Yaskawa INFORM job: FMTV_HOOD_FASH.JBI

/JOB
//NAME FMTV_HOOD_FASH
//POS
///NPOS 40,0,0,0,0,0
///TOOL 0
///POSTYPE PULSE
///PULSE
C00000=-63952,-155163,126853,-105316,-81596,-126671
C00001=-64461,-165808,55284,-105319,-116136,-134897
C00002=-65360,-175099,-71284,-105325,-123848,-149443
C00003=16523,-162142,-76585,-105325,-105920,-149443
C00004=136824,-41147,-71653,-105908,-92109,-42430
C00005=136265,2790,-33985,-105635,-93453,-40514
C00006=131512,-1858,-30509,-105042,-95515,-43185
C00007=137993,-15449,-40810,-106144,-90722,-43513
C00008=137236,-27294,-42795,-96614,-65040,-40742
C00009=140665,-37218,-47628,-99236,-35066,-29992
C00010=140875,-41659,-45027,-77194,-30549,-37243
C00011=146366,-51964,-56030,-75285,-24000,-39354
C00012=156119,-65002,-57409,-21147,-27778,-71904
C00013=185515,-90979,-56740,15089,-40881,-92836
C00014=189457,-94504,-56572,18214,-43459,-94468
C00015=185283,-96154,-47186,13023,-48087,-91295
C00016=200345,-105201,-46417,22564,-56140,-91888
C00017=216925,-109654,-49443,33869,-61566,-97373
C00018=254335,-111877,-36308,-709,-80515,-94448
C00019=248884,-122551,-45515,-3659,-81498,-92809
C00020=231141,-122690,-119580,-13159,-82300,-87441
C00021=-123049,-84648,-100330,119939,-63154,47192
C00022=-145736,-60124,-89141,132014,-54215,37600
C00023=-142792,-13464,-52848,133356,-59585,35650
C00024=-142664,-20455,-52488,131545,-57125,37514
C00025=-150130,-32967,-58116,133370,-50891,37010
C00026=-145449,-39905,-51845,93454,-46937,51672
C00027=-145191,-39750,-50505,88326,-47662,51868
C00028=-144160,-44267,-45166,62771,-52773,58710
C00029=-148791,-53730,-48823,49689,-54914,64885
C00030=-150743,-57181,-50382,48425,-54527,66002
C00031=-175825,-83730,-45254,23478,-63050,83138
C00032=-177177,-85796,-44891,22474,-63852,83945
C00033=-172411,-84272,-42490,25021,-65496,77234
C00034=-167210,-84468,-34339,27016,-70739,76523
C00035=-180047,-97470,-37743,19473,-72177,81934
C00036=-191369,-102527,-40604,12946,-71396,85928
C00037=-242211,-114344,-41149,18289,-76989,98255
C00038=-243523,-126027,-51318,17488,-77632,98803
C00039=-252640,-156391,-84960,58658,-32345,33822
//INST
///DATE 2023/09/19 14:49
///ATTR SC,RW
///GROUP1 RB1
NOP
MOVJ C00000 VJ=65.00  //HOME
MOVJ C00001 VJ=65.00
MOVJ C00002 VJ=65.00  //ROTATE
MOVJ C00003 VJ=65.00
MOVJ C00004 VJ=65.00
MOVL C00005 V=150.0  //OVER
MOVL C00006 V=100.0  //UP TO
MOVL C00007 V=25.0  //INTO
MOVL C00008 V=25.0
MOVL C00009 V=25.0
MOVL C00010 V=25.0
MOVL C00011 V=25.0
MOVL C00012 V=25.0
MOVL C00013 V=25.0
MOVL C00014 V=25.0
MOVL C00015 V=25.0
MOVL C00016 V=25.0
MOVL C00017 V=25.0
MOVL C00018 V=25.0  //END
MOVL C00019 V=45.0  //OUT
MOVJ C00020 VJ=65.00
MOVJ C00021 VJ=65.00
MOVL C00022 V=65.0
MOVL C00023 V=65.0
MOVL C00024 V=65.0  //INLINE
MOVL C00025 V=25.0
MOVL C00026 V=25.0  //CORNER
MOVL C00027 V=10.0
MOVL C00028 V=25.0
MOVL C00029 V=25.0
MOVL C00030 V=25.0
MOVL C00031 V=25.0
MOVL C00032 V=25.0
MOVL C00033 V=25.0
MOVL C00034 V=25.0
MOVL C00035 V=25.0
MOVL C00036 V=25.0
MOVL C00037 V=25.0  //END
MOVJ C00038 VJ=65.00
MOVJ C00039 VJ=65.00  //AWAY
END
